INTERFACE I_Navitrol_OmniDriveMotorControl EXTENDS I_Base

END_INTERFACE

(* stored: Version 1.1.0.1
   Itf I_Navitrol_OmniDriveMotorControl: Id {1fbfdd5b-d5a6-4d0d-8de7-eec24baec004} *)
